// TIA Portal V18 export
TYPE "Console_IO_In"
   STRUCT
      Slot1 { S7_SetPoint := 'True'} : "DI16x24V_In";
      Slot2 { S7_SetPoint := 'True'} : "DI16x24V_In";
      Slot3 { S7_SetPoint := 'True'} : "AI8xU_In";
   END_STRUCT;
END_TYPE
